INTERFACE ITF_Podzespol

PROPERTY Bazowanie : BOOL
GET
END_GET
END_PROPERTY

PROPERTY Bazuj : BOOL
SET
END_SET
END_PROPERTY

METHOD CyklBazowania_Praca : BOOL
VAR_INPUT
END_VAR
END_METHOD

PROPERTY CyklPracy : BOOL
GET
END_GET
END_PROPERTY

METHOD CyklPracy_Praca : BOOL
VAR_INPUT
END_VAR
END_METHOD

PROPERTY CyklPracySkonczony : BOOL
GET
END_GET
END_PROPERTY

METHOD Praca : BOOL
VAR_INPUT
END_VAR
END_METHOD

METHOD Resetowanie : BOOL
VAR_INPUT
END_VAR
END_METHOD

PROPERTY Resetuj : BOOL
SET
END_SET
END_PROPERTY

PROPERTY WykonajCyklPracy : BOOL
SET
END_SET
END_PROPERTY

END_INTERFACE

(* stored: Version 1.1.0.1, ProductVersion 3.1.4024.11
   Itf ITF_Podzespol: Id {5d25e72b-1438-44c3-b36e-0885f28d066d}
   Property Bazowanie: Id {7b397dae-2a67-4c52-821b-2d0d89e6efc0}
   Get Get: Id {55a70d2c-7ef8-4aa0-9600-fd519c399e36}
   Property Bazuj: Id {15e4b681-3893-4eaa-8788-a93fd0efaee4}
   Set Set: Id {c735cbdf-f000-4512-ac9b-366d8d190dcb}
   Method CyklBazowania_Praca: Id {d632d771-9980-4097-9c77-aee8c894d905}
   Property CyklPracy: Id {bfb099a0-998b-4882-8686-2985e13b715b}
   Get Get: Id {b49a6731-cfb1-453c-ab0e-40d4e9384c2f}
   Method CyklPracy_Praca: Id {bb6f835d-1ae3-49a1-afa3-7f7c9567a0e6}
   Property CyklPracySkonczony: Id {3772dc0e-11a7-4714-8bd5-32cd4c030af3}
   Get Get: Id {c87ffec6-e3fe-4163-aaed-359f74bb4295}
   Method Praca: Id {cdd1443e-4aef-41f9-8ae1-db2e9e1959a0}
   Method Resetowanie: Id {2cc9d381-ed8d-4245-a9b7-dee98be1f3f8}
   Property Resetuj: Id {ed86aa34-1e7f-448e-b4eb-efd94c830e9c}
   Set Set: Id {5ec24030-3ae1-4862-8d44-ef9b0e14ed88}
   Property WykonajCyklPracy: Id {cdeb26fc-e3db-4305-9597-6cc3c95009ce}
   Set Set: Id {ed12fddf-61cb-4d2a-a301-ed247672199c} *)
